RoboDK station: AGameOfChess.rdk

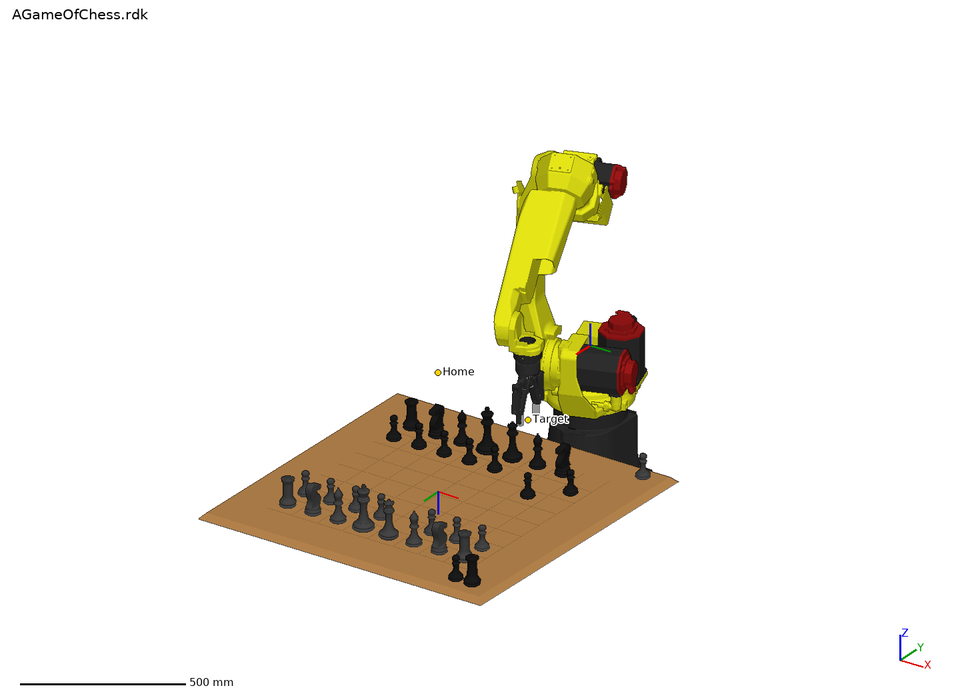
[picture v0: the station drawn from its stored meshes, robots at their saved joint values, targets as dots, program paths as lines]
Station AGameOfChess (saved by RoboDK 5.5.1). Poses are relative to the parent item; angles as X-Y-Z fixed-axis rotations.
  - frame Fanuc M-10iA Base at (0, 800, 180) mm, rotated rx 0 ry 0 rz -90 deg
    - robot Fanuc M-10iA: 6 axes, payload 10 kg, reach 1420 mm, repeatability 0.08 mm, weight 130 kg
        modified DH rows (alpha deg, a mm, theta deg, d mm): 0, 0, 0, 450; -90, 150, -90, 0; 0, 600, 0, 0; -90, 200, 0, 640; 90, 0, 0, 0; -90, 0, 0, 100
        base shift (0, 0, -450) mm
        joint limits [-180, -90, -95, -190, -190, -360] to [180, 160, 180, 190, 190, 360]; home [0, 0, 0, 0, 0, 0]; saved at [19.367, -8.158, -36.16, 0, -53.84, -19.367]
      - tool RobotiQ 2F-140 Gripper (Open), TCP at (0, 0, 200) mm, size 139 x 75 x 203.7 mm
      - tool RobotiQ 2F-140 Gripper (Closed), TCP at (0, 0, 200) mm, size 124 x 75 x 244.3 mm
    - frame ZeroPoint at (800, 0, -172.22) mm, rotated rx 180 ry 0 rz 90 deg
      - target Home (Cartesian target) at (0, 0, -400) mm; joints [0, 17.552, -21.141, 0, -68.859, 90] of Fanuc M-10iA
      - target Target (Cartesian target) at (232, -140, -250) mm, rotated rx 0 ry 0 rz 90 deg; joints [29.841, 9.478, -35.968, 0, -54.032, -29.841] of Fanuc M-10iA
  - folder Schwarz_Spielfiguren
    - object sBauer at (-465, -93, 0) mm, size 48.6 x 82.2 x 48.6 mm, geometry from sBauer.glb
    - object sBauer at (-558, -93, 0) mm, size 48.6 x 82.2 x 48.6 mm, geometry from sBauer.glb
    - object sLaeufer at (-186, 0, 0) mm, size 52.8 x 115.2 x 52.7 mm, geometry from sLaeufer.glb
    - object sBauer at (-279, -93, 0) mm, size 48.6 x 82.2 x 48.6 mm, geometry from sBauer.glb
    - object sBauer at (-651, -93, 0) mm, size 48.6 x 82.2 x 48.6 mm, geometry from sBauer.glb
    - object sLaeufer at (-465, 0, 0) mm, size 52.8 x 115.2 x 52.7 mm, geometry from sLaeufer.glb
    - object 5_sBauer at (-372, -93, 0) mm, size 48.6 x 82.2 x 48.6 mm, geometry from sBauer.glb
    - object sBauer at (0, -93, 0) mm, size 48.6 x 82.2 x 48.6 mm, geometry from sBauer.glb
    - object sSpringer at (-558, 0, 0) mm, size 52.8 x 104.4 x 52.8 mm, geometry from sSpringer.glb
    - object sSpringer at (-93, 0, 0) mm, size 52.8 x 104.4 x 52.8 mm, geometry from sSpringer.glb
    - object sTurm at (-651, 0, 0) mm, size 52.7 x 95.3 x 52.8 mm, geometry from sTurm.glb
    - object sKoenig at (-372, 0, 0) mm, size 70.2 x 151 x 70.2 mm, geometry from sKoenig.glb
    - object sDame at (-279, 0, 0) mm, size 62.6 x 128.5 x 62.5 mm, geometry from sDame.glb
  - folder Weisse_Spielfiguren
    - object wBauer at (-372, -558, 0) mm, size 48.6 x 82.2 x 48.6 mm, geometry from wBauer.glb
    - object wBauer at (-465, -558, 0) mm, size 48.6 x 82.2 x 48.6 mm, geometry from wBauer.glb
    - object wBauer at (-651, -558, 0) mm, size 48.6 x 82.2 x 48.6 mm, geometry from wBauer.glb
    - object wLaeufer at (-186, -651, 0) mm, size 52.8 x 115.2 x 52.7 mm, geometry from wLaeufer.glb
    - object wLaeufer at (-465, -651, 0) mm, size 52.8 x 115.2 x 52.7 mm, geometry from wLaeufer.glb
    - object wBauer at (0, -558, 0) mm, size 48.6 x 82.2 x 48.6 mm, geometry from wBauer.glb
    - object wBauer at (-558, -558, 0) mm, size 48.6 x 82.2 x 48.6 mm, geometry from wBauer.glb
    - object wSpringer at (-558, -651, 0) mm, size 52.8 x 104.4 x 52.8 mm, geometry from wSpringer.glb
    - object wBauer at (-93, -558, 0) mm, size 48.6 x 82.2 x 48.6 mm, geometry from wBauer.glb
    - object wBauer at (-186, -558, 0) mm, size 48.6 x 82.2 x 48.6 mm, geometry from wBauer.glb
    - object wSpringer at (-93, -651, 0) mm, size 52.8 x 104.4 x 52.8 mm, geometry from wSpringer.glb
    - object wTurm at (0, -651, 0) mm, size 52.7 x 95.3 x 52.8 mm, geometry from wTurm.glb
    - object wTurm at (-651, -651, 0) mm, size 52.7 x 95.3 x 52.8 mm, geometry from wTurm.glb
    - object wKoenig at (-372, -651, 0) mm, size 70.2 x 151 x 70.2 mm, geometry from wKoenig.glb
    - object wDame at (-279, -651, 0) mm, size 62.6 x 128.5 x 62.5 mm, geometry from wDame.glb
  - program main (7 instructions, listed below)
  - Python program tcpIPServer (listed below)
  - program AttachFigure (3 instructions, listed below)
  - program DetachFigure (3 instructions, listed below)
  - object Spielbrett at (0, 0, 0) mm, size 1041 x 20.5 x 1041 mm, geometry from Spielbrett.glb
    - object sTurm at (115, -775, 0) mm, size 52.7 x 95.3 x 52.8 mm, geometry from sTurm.glb
    - object sBauer at (55, -775, 0) mm, size 48.6 x 82.2 x 48.6 mm, geometry from sBauer.glb
    - object wBauer at (115, 124, 0) mm, size 48.6 x 82.2 x 48.6 mm, geometry from wBauer.glb
    - object sBauer at (-93, -185, 0) mm, size 48.6 x 82.2 x 48.6 mm, geometry from sBauer.glb

--- program main (robot Fanuc M-10iA) ---
  Referenz erstellen.: ZeroPoint
  Werkzeug setzen: RobotiQ 2F-140 Gripper (Open)
  Objekte ersetzen
  MoveJ (Home)
  Anzeigen RobotiQ 2F-140 Gripper (Open)
  Verstecken RobotiQ 2F-140 Gripper (Closed)
  Aufruf tcpIPServer

--- Python program tcpIPServer ---
from robodk import *  # RoboDK API
from robodk import *   # Robot toolbox
RDK = robolink.Robolink()

import socket

HOST = "127.0.0.1"
PORT = 65432

robot = RDK.Item('Fanuc M-10iA')
target = RDK.Item('Target')
"""
while(True):
    target.setPose(KUKA_2_Pose([773, 232, 0, 90, 0, 180]))
    robot.MoveJ(target);
    target.setPose(KUKA_2_Pose([680, 325, 0, 90, 0, 180]))
    robot.MoveJ(target);

"""
with socket.socket(socket.AF_INET, socket.SOCK_STREAM) as s:
    s.bind((HOST, PORT))
    s.listen()
    conn, addr = s.accept()
    with conn:
        response = "done\n";
        conn.sendall(bytes(response, 'utf-8'))
        while True:
            data = conn.recv(1024)
            if not data:
                break

            dataPos = data.decode('utf-8').split(';')
            target.setPose(KUKA_2_Pose([int(dataPos[0]), int(dataPos[1]), -250, 90, 0, 0]))
            robot.MoveJ(target);
            target.setPose(KUKA_2_Pose([int(dataPos[0]), int(dataPos[1]), -80, 90, 0, 0]))
            robot.MoveL(target);
            RDK.Item(dataPos[2]).RunProgram()
            target.setPose(KUKA_2_Pose([int(dataPos[0]), int(dataPos[1]), -250, 90, 0, 0]))
            robot.MoveL(target);

            response = "done\n";
            conn.sendall(bytes(response, 'utf-8'))

--- program AttachFigure (robot Fanuc M-10iA) ---
  Anzeigen RobotiQ 2F-140 Gripper (Closed)
  Verstecken RobotiQ 2F-140 Gripper (Open)
  Anhängen an RobotiQ 2F-140 Gripper (Open)

--- program DetachFigure (robot Fanuc M-10iA) ---
  Anzeigen RobotiQ 2F-140 Gripper (Open)
  Verstecken RobotiQ 2F-140 Gripper (Closed)
  Ablösen von RobotiQ 2F-140 Gripper (Open)
